FUNCTION_BLOCK POU
VAR_INPUT
END_VAR
VAR_OUTPUT
END_VAR
VAR
	AddTwo: INT;
END_VAR

END_FUNCTION_BLOCK

(* stored: Version 1.1.0.1, ProductVersion 3.1.4024.6
   POU POU: Id {cf36082a-cd52-4292-96c2-0560cba85e60}, SpecialFunc None *)
